// TIA Portal V19 export
TYPE "LEXCHANGETRAY_typeVfd_controlInterface"
// stored: Access Published
   STRUCT
      cmd : "LEXCHANGETRAY_typeVfd_cmd";
      par : "LEXCHANGETRAY_typeVfd_par";
      monitor : "LEXCHANGETRAY_typeVfd_monitor";
      Config : "LBC_typeSinaSpeedConfiguration";
      sinaControlNode { S7_SetPoint := 'True'} : "LBC_typeSinaSpeedControlNode";
   END_STRUCT;
END_TYPE
